FUNCTION_BLOCK DOSomething
VAR_INPUT
	input :BOOL;
END_VAR
VAR_OUTPUT
END_VAR
VAR
	isDoorOpen : BOOL;
END_VAR

IF isDoorOpen THEN
	//
END_IF

METHOD method1 : BOOL
VAR_INPUT
END_VAR
VAR
	currentAlarm1State : machineStates;
	currentAlarm2State : machineStates;
END_VAR
//do something
case
END_METHOD

END_FUNCTION_BLOCK

(* stored: Version 1.1.0.1, ProductVersion 3.1.4024.12
   POU DOSomething: Id {0057b8ad-0eae-4e90-bfb0-21f4dbb3901e}, SpecialFunc None
   Method method1: Id {de18747c-8189-46bb-bf3e-9c8d890715bd} *)
